PROGRAM Prg_MainCall

Prg.MainCall();

END_PROGRAM

(* stored: Version 1.1.0.1
   POU Prg_MainCall: Id {89223677-ca7f-4e78-9fc2-b5acd4173a8f}, SpecialFunc None *)
